{attribute 'no_explicit_call' := 'do not call this function block directly'} 
{attribute 'enable_dynamic_creation'}
FUNCTION_BLOCK DictionaryEnumerator EXTENDS Object IMPLEMENTS IEnumerator
VAR
	_ClassName : STRING := __POUNAME();
	
	_Dictionary : IReadOnlyDictionary;
	_CurrentIndex : DINT := -1;
END_VAR

{attribute 'monitoring' := 'call'}
PROPERTY ClassName : STRING
GET
ClassName := _ClassName;
END_GET
END_PROPERTY

// Shows curent collection element
PROPERTY Current : PVOID
GET
VAR
	genericValue : REFERENCE TO GENERIC_KEY_VALUE_PAIR;
END_VAR
IF _CurrentIndex >= 0 AND_THEN _CurrentIndex < _Dictionary.Count THEN
	genericValue REF= _Dictionary.GetKeyValuePairByIndex(_CurrentIndex); 
	Current := ADR(genericValue);
ELSE
	Current := 0;	
END_IF
END_GET
END_PROPERTY

PROPERTY CurrentValue : REFERENCE TO GENERIC_KEY_VALUE_PAIR
GET
VAR
	valuePointer : POINTER TO GENERIC_KEY_VALUE_PAIR;
END_VAR
valuePointer := Current;

IF valuePointer <> 0 THEN
	CurrentValue REF= valuePointer^;	
END_IF
END_GET
END_PROPERTY

METHOD FB_init : BOOL
VAR_INPUT
	(* if TRUE, the retain variables are initialized (warm start / cold start)*)
	bInitRetains	: BOOL;
	(* if TRUE, the instance afterwards gets moved into the copy code (online change)*)
	bInCopyCode	: BOOL;
	dictionary : IReadOnlyDictionary;
END_VAR
_Dictionary := dictionary;
END_METHOD

{attribute "object_name" := "MoveNext"}
METHOD MoveNext : BOOL
_CurrentIndex := _CurrentIndex + 1;

MoveNext := _CurrentIndex < _Dictionary.Count;
END_METHOD

{attribute "object_name" := "Reset"}
METHOD Reset
_CurrentIndex := -1;
END_METHOD

{attribute 'monitoring' := 'call'}
PROPERTY Size : ULINT
GET
Size := XSIZEOF(THIS^);
END_GET
END_PROPERTY

END_FUNCTION_BLOCK

(* stored: Version 1.1.0.1
   POU DictionaryEnumerator: Id {2f365963-7036-4f79-8584-bc80ea1e769d}, SpecialFunc None
   Property ClassName: Id {839d6121-03b1-4336-9ccf-f78a04cd0cb5}
   Get Get: Id {e0aa9b3a-9a64-4398-b874-5ed4b802f8a8}
   Property Current: Id {9d7a3084-f2d9-46a4-babc-c0d4307e4c92}
   Get Get: Id {f0a9af6e-a818-4733-9637-b26e3a47ceb1}
   Property CurrentValue: Id {a11fa9ca-d7fd-47e7-8c94-382211eba30f}
   Get Get: Id {587ce946-29e3-488a-a34c-6505b64fa177}
   Method FB_init: Id {5f1ac79b-7b16-408a-a050-ca6526d9c743}
   Method MoveNext: Id {a3b96f77-158c-4502-97c9-c508c77c0dd2}
   Method Reset: Id {ffc13050-106a-4a43-ad03-55630a53602f}
   Property Size: Id {1db19b22-0572-4a68-948e-fa84d0bb1deb}
   Get Get: Id {ee09e011-6acd-46b1-94f4-d278acd0fb55} *)
